TYPE ST_Inverter_additionalTemperatures :
STRUCT
	r_ambient					: REAL;
	r_CMchokeOuter				: ARRAY[1..4] OF REAL;
	r_CMchokeInner				: ARRAY[1..4] OF REAL;
	r_GrChokeOuter				: ARRAY[1..3] OF REAL;
	r_GrChokeInner				: ARRAY[1..3] OF REAL;
	r_ACCapsTop					: REAL;
	r_ACCapsBottom				: REAL;
	r_DCCaps					: REAL;
	r_ACbusbarOutput			: REAL;
	r_ACbusbarCMchoke			: REAL;
	r_DCbusbarCMChoke			: REAL;
	r_AirInletModule			: REAL;
	r_AirOutletFancoil			: REAL;
	r_WaterInletFancoil			: REAL;
	r_WaterOutletFancoil		: REAL;
	r_FancoilCompartement		: REAL;
END_STRUCT
END_TYPE

(* stored: Version 1.1.0.1, ProductVersion 3.1.4026.18
   DUT ST_Inverter_additionalTemperatures: Id {1c232955-9130-41ad-af2a-60df0dd2eb44} *)
